SYSTEM testThreads (* System Configuration *)
  (* Standard: 61499-1 *)
  (* Version 0.3, 2003-12-05, JHC, Rockwell Automation, Renamed from NEWSYSTEM. *)
  (* Version 0.2, 2002-11-05, JHC, Rockwell Automation, Fixed missing (empty) FBD in Application. *)
  (* Version 0.1, 2002-01-17, JHC, Rockwell Automation, Minor cleanup *)
  (* Version 0.0, 2000-05-27, JHC, Rockwell Automation *)
  APPLICATION APP1
  END_APPLICATION
  DEVICE DEV1 : DeviceType
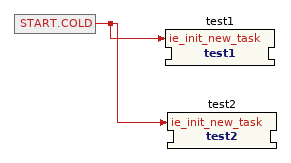
    [picture p0: device DEV1]
    FBS
      test1 : test1;
      test2 : test2;
    END_FBS
    EVENT_CONNECTIONS
      START.COLD TO test1.ie_init_new_task;
      START.COLD TO test2.ie_init_new_task;
    END_CONNECTIONS
  END_DEVICE
END_SYSTEM
